// TIA Portal V19 export
FUNCTION_BLOCK "WeeklyClock"   // FB84, LAD
TITLE = WEEKLY CLOCK MANAGEMENT
// stored: Access Published, MemoryReserve 100, SetENOAutomatically false
   VAR_INPUT
      DaySetup : Array[1..7] of "WkClockSet";   // 1=Sunday...7=Saturday
      CabinetCooling : "WkClockSet";
      ClockEnable : Bool;
      CabinetCoolingEnable : Bool;
   END_VAR
   VAR_OUTPUT
      ClockActive : Bool;
      CabinetCoolingActive : Bool;
   END_VAR
   VAR DB_SPECIFIC
      ActualDT : DTL;
      ActualTime : Time_Of_Day;
      ActualDate : Date;
      ActuaDtON : DTL;
      ActualDtOFF : DTL;
      DayEnable : Array[1..7] of Bool;   // 1=Sunday...7=Saturday
      CabinetEnable : Bool;
   END_VAR
   VAR_TEMP
      retVal : Int;
      IsGt : Bool;
      IsLt : Bool;
      TimeOfD : Time_Of_Day;
   END_VAR
BEGIN

REGION Network 1: Get actual date and time
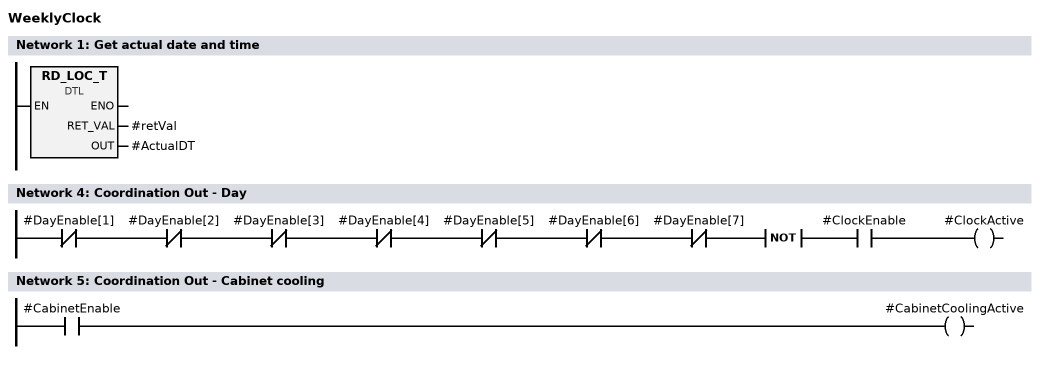
   RUNG wire#powerrail
      { S7_Templates := "date_type := DTL" } RD_LOC_T(RET_VAL => #retVal, OUT => #ActualDT)
   END_RUNG
   // the same network as SCL:
   #retVal := RD_LOC_T(OUT => #ActualDT);
END_REGION

REGION Network 2 (SCL): Days of week for oil Heating
   #ActualDate := DTL_TO_DATE(#ActualDT);
   #ActuaDtON := CONCAT_DATE_TOD(IN1 := #ActualDate, IN2 := #DaySetup[#ActualDT.WEEKDAY].Set_ON);
   #ActualDtOFF := CONCAT_DATE_TOD(IN1 := #ActualDate, IN2 := #DaySetup[#ActualDT.WEEKDAY].Set_OFF);
   #IsGt := #ActualDT >= #ActuaDtON;
   #IsLt := #ActualDT <= #ActualDtOFF;

   #DayEnable[#ActualDT.WEEKDAY] := #IsGt AND #IsLt AND #DaySetup[#ActualDT.WEEKDAY].Enable;
END_REGION

REGION Network 3 (SCL): Cabinet cooling
   #ActualDate := DTL_TO_DATE(#ActualDT);
   #ActuaDtON := CONCAT_DATE_TOD(IN1 := #ActualDate, IN2 := #CabinetCooling.Set_ON);
   #ActualDtOFF := CONCAT_DATE_TOD(IN1 := #ActualDate, IN2 := #CabinetCooling.Set_OFF);
   #IsGt := #ActualDT >= #ActuaDtON;
   #IsLt := #ActualDT <= #ActualDtOFF;

   #CabinetEnable := #IsGt AND #IsLt AND #CabinetCooling.Enable;
END_REGION

REGION Network 4: Coordination Out - Day
   RUNG wire#powerrail
      I_Contact( #DayEnable[1] )
      I_Contact( #DayEnable[2] )
      I_Contact( #DayEnable[3] )
      I_Contact( #DayEnable[4] )
      I_Contact( #DayEnable[5] )
      I_Contact( #DayEnable[6] )
      I_Contact( #DayEnable[7] )
      Not()
      Contact( #ClockEnable )
      Coil( #ClockActive )
   END_RUNG
   // the same network as SCL:
   #ClockActive := NOT (NOT #DayEnable[1] AND NOT #DayEnable[2] AND NOT #DayEnable[3] AND NOT #DayEnable[4] AND NOT #DayEnable[5] AND NOT #DayEnable[6] AND NOT #DayEnable[7]) AND #ClockEnable;
END_REGION

REGION Network 5: Coordination Out - Cabinet cooling
   RUNG wire#powerrail
      Contact( #CabinetEnable )
      Coil( #CabinetCoolingActive )
   END_RUNG
   // the same network as SCL:
   #CabinetCoolingActive := #CabinetEnable;
END_REGION
END_FUNCTION_BLOCK
